SUBAPPLICATION Uebung_090a2 (* Beispiel für F_MUX_3 *)
  (* Standard: 61499-2; Description: Copyright (c) 2023 Meisterschulen am Ostbahnhof This program and the accompanying materials are made available under the terms of the Eclipse Public License 2.0 which is available at https://www.eclipse.org/legal/epl-2.0/ SPDX-License-Identifier: EPL-2.0 *)
  (* Version 1.0, 2023-10-23, Franz Höpfinger, Meisterschulen am Ostbahnhof *)
  IMPORT logiBUS::io::DI::logiBUS_DI;
  IMPORT logiBUS::io::DI::logiBUS_DI_Events;
  IMPORT logiBUS::io::DQ::logiBUS_DO;
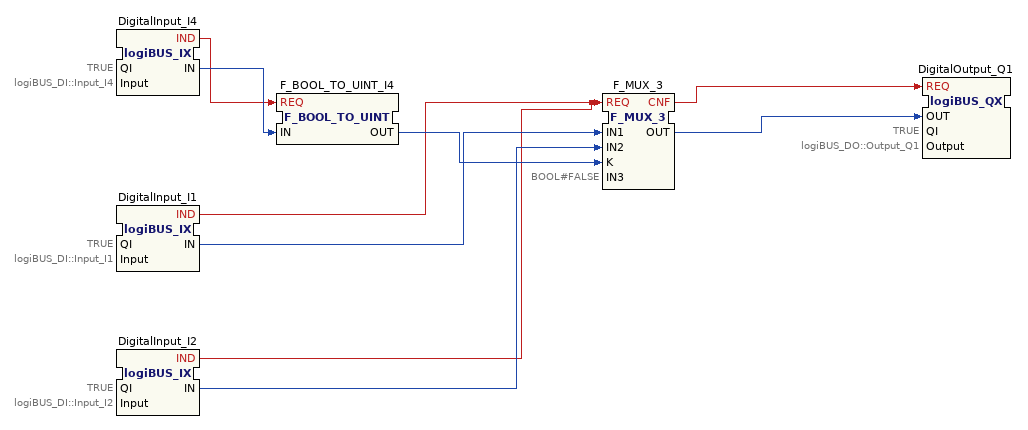
  (* BROKEN ! diese Übung lässt sich nicht aufspielen ! https://github.com/eclipse-4diac/4diac-forte/issues/324 *)
  FBS
    F_MUX_3 : F_MUX_3(IN3 := BOOL#FALSE);
    DigitalInput_I4 : logiBUS::io::DI::logiBUS_IX(QI := TRUE, Input := logiBUS_DI::Input_I4);
    F_BOOL_TO_UINT_I4 : F_BOOL_TO_UINT;
    DigitalOutput_Q1 : logiBUS::io::DQ::logiBUS_QX(QI := TRUE, Output := logiBUS_DO::Output_Q1);
    DigitalInput_I1 : logiBUS::io::DI::logiBUS_IX(QI := TRUE, Input := logiBUS_DI::Input_I1);
    DigitalInput_I2 : logiBUS::io::DI::logiBUS_IX(QI := TRUE, Input := logiBUS_DI::Input_I2);
  END_FBS
  EVENT_CONNECTIONS
    DigitalInput_I4.IND TO F_BOOL_TO_UINT_I4.REQ;
    F_MUX_3.CNF TO DigitalOutput_Q1.REQ;
    DigitalInput_I1.IND TO F_MUX_3.REQ;
    DigitalInput_I2.IND TO F_MUX_3.REQ;
  END_CONNECTIONS
  DATA_CONNECTIONS
    F_MUX_3.OUT TO DigitalOutput_Q1.OUT;
    DigitalInput_I1.IN TO F_MUX_3.IN1;
    DigitalInput_I2.IN TO F_MUX_3.IN2;
    DigitalInput_I4.IN TO F_BOOL_TO_UINT_I4.IN;
    F_BOOL_TO_UINT_I4.OUT TO F_MUX_3.K;
  END_CONNECTIONS
END_SUBAPPLICATION
